# EPICS autosave request: opticsApp/Db/kohzuSeq_settings.req
# Kohzu monochromator
$(P)BraggHAO.VAL
$(P)BraggKAO.VAL
$(P)BraggLAO.VAL
$(P)BraggAAO.VAL
$(P)BraggTypeMO.VAL
$(P)KohzuMode2MO.VAL
$(P)Kohzu_yOffsetAO.VAL
$(P)KohzuSpeedCtrl
